FUNCTION_BLOCK FB_T1_InputSource IMPLEMENTS I_InputSource
VAR
	_eDataState: E_DataSourceState;
	
	_nMaxOversamplingFactor: UDINT := 1;
	
	_nElements: UDINT;
	_nCurrentElement: UDINT;
	_nDataHandle: ULINT;
	
	_nClientListHash: LWORD;
	_nCurrentClientHash: LWORD;
	
	_stInputs: ST_T1_Inputs;
	
	fbIotSymbol_GVL_Components_fbMachine_stAnalytics_nState: FB_ALY_IotSymbol_UINT := (stConfig:= (sSymbolName:= 'GVL_Components.fbMachine.stAnalytics.nState'));
	fbIotSymbol_GVL_Components_fbMachine_stAnalytics_nUnitsProduced: FB_ALY_IotSymbol_ULINT := (stConfig:= (sSymbolName:= 'GVL_Components.fbMachine.stAnalytics.nUnitsProduced'));
	fbIotSymbol_GVL_Components_fbMachine_stAnalytics_nDefectiveUnits: FB_ALY_IotSymbol_ULINT := (stConfig:= (sSymbolName:= 'GVL_Components.fbMachine.stAnalytics.nDefectiveUnits'));
	fbIotSymbol_GVL_Components_fbMachine_stAnalytics_tMlCalculation: FB_ALY_IotSymbol_UDINT := (stConfig:= (sSymbolName:= 'GVL_Components.fbMachine.stAnalytics.tMlCalculation'));
	
	//Target T1 = Broker:"localhost" Topic:"DefaultMainTopic/PlcStream1"
	fbStreamHelper: FB_ALY_StreamHelper;
	bConfigured: BOOL := FALSE;
	
	fbTON_DataTimeout: TON;
END_VAR
VAR_STAT
	_nClientIndex: INT;
END_VAR

METHOD AddClient : BOOL
VAR_OUTPUT
	nClientID: LWORD;
END_VAR
VAR
END_VAR
nClientID:= TO_LWORD(EXPT(2,_nClientIndex));
_nClientIndex:= _nClientIndex + 1;

_nClientListHash:= _nClientListHash + nClientID;
END_METHOD

PROPERTY bReadNewData : BOOL
GET
bReadNewData:= _nElements = 0 OR _nCurrentClientHash >= _nClientListHash;
END_GET
END_PROPERTY

METHOD Call : BOOL
VAR
	stConfig: ST_ALY_StreamHelper_Config;
END_VAR
IF NOT fbStreamHelper.bConfigured THEN
	stConfig.nObjectID:= 16#01010110;
	stConfig.nNumInputBuffer:= 20;
	fbStreamHelper.Configure(stConfig);
END_IF

IF NOT bConfigured THEN
	//GVL_Components.fbMachine.stAnalytics.nState
	fbStreamHelper.AddIotSymbol(fbIotSymbol_GVL_Components_fbMachine_stAnalytics_nState);
	//GVL_Components.fbMachine.stAnalytics.nUnitsProduced
	fbStreamHelper.AddIotSymbol(fbIotSymbol_GVL_Components_fbMachine_stAnalytics_nUnitsProduced);
	//GVL_Components.fbMachine.stAnalytics.nDefectiveUnits
	fbStreamHelper.AddIotSymbol(fbIotSymbol_GVL_Components_fbMachine_stAnalytics_nDefectiveUnits);
	//GVL_Components.fbMachine.stAnalytics.tMlCalculation
	fbStreamHelper.AddIotSymbol(fbIotSymbol_GVL_Components_fbMachine_stAnalytics_tMlCalculation);

	bConfigured:= TRUE;
END_IF

fbStreamHelper.Call();
IF fbStreamHelper.bError THEN
	_eDataState:= E_DataSourceState.eError;
ELSIF NOT fbStreamHelper.bConnected THEN
	_eDataState:= E_DataSourceState.eNotConnected;
ELSE
	_nElements:= fbStreamHelper.nNumElements;
	IF _nElements > 0 THEN
		_eDataState:= E_DataSourceState.eReceiveData;
	END_IF

	fbTON_DataTimeout(IN:= _nElements = 0, PT:= T#5S);
	IF fbTON_DataTimeout.Q THEN
		_eDataState:= E_DataSourceState.eWaitForData;
	END_IF
END_IF

IF _nElements > 0 THEN
	_nDataHandle:= _nDataHandle + 1;
	_nCurrentClientHash:= 0;
END_IF

_nCurrentElement:= 0;
END_METHOD

METHOD ClientDone : BOOL
VAR_INPUT
	nClientID: LWORD;
END_VAR
VAR
END_VAR
_nCurrentClientHash:=  _nCurrentClientHash + nClientID;
END_METHOD

PROPERTY eDataState : E_DataSourceState
GET
eDataState:= _eDataState;
END_GET
END_PROPERTY

METHOD GetData : BOOL
VAR_INPUT
	nElement: UDINT;
	pInputs: PVOID;
	nInputsSize: UDINT;
END_VAR
VAR_OUTPUT
	nTimestamp: ULINT;
	nContext: DWORD;
END_VAR
VAR
	_nElement: UDINT;
	_pInputs: PVOID;
	_nInputsSize: UDINT;
END_VAR
Analytics.fbT1_IecCriticalSection.Enter();

_nElement:= nElement;
_pInputs:= pInputs;
_nInputsSize:= nInputsSize;

nContext:= 0;
IF nElements > 0 THEN
	IF _nElement <= nElements THEN

		IF _nCurrentElement <> _nElement THEN

			//Set local raw inputs
			_stInputs.nGVL_Components_fbMachine_stAnalytics_nState:= fbIotSymbol_GVL_Components_fbMachine_stAnalytics_nState.GetValue(_nElement);
			_stInputs.nGVL_Components_fbMachine_stAnalytics_nUnitsProduced:= fbIotSymbol_GVL_Components_fbMachine_stAnalytics_nUnitsProduced.GetValue(_nElement);
			_stInputs.nGVL_Components_fbMachine_stAnalytics_nDefectiveUnits:= fbIotSymbol_GVL_Components_fbMachine_stAnalytics_nDefectiveUnits.GetValue(_nElement);
			_stInputs.nGVL_Components_fbMachine_stAnalytics_tMlCalculation:= fbIotSymbol_GVL_Components_fbMachine_stAnalytics_tMlCalculation.GetValue(_nElement);

			nContext:= E_DataSourceContext.eContext_1000;
			_nCurrentElement:= _nElement;
		END_IF

		//Set output values
		IF _pInputs > 0 THEN
			MEMCPY(_pInputs, ADR(_stInputs), _nInputsSize);
			nTimestamp:= fbStreamHelper.GetTimestampElement(_nElement);
		END_IF
	END_IF
	GetData:= TRUE;
ELSE
	GetData:= FALSE;
END_IF

Analytics.fbT1_IecCriticalSection.Leave();
END_METHOD

PROPERTY nDataHandle : ULINT
GET
nDataHandle:= _nDataHandle;
END_GET
END_PROPERTY

PROPERTY nElements : UDINT
GET
nElements:= _nElements;
END_GET
END_PROPERTY

METHOD NewDataAvailable : BOOL
VAR_INPUT
	nLastDataHandle: ULINT;
END_VAR
VAR
END_VAR
NewDataAvailable:= _nElements > 0 AND _nDataHandle <> nLastDataHandle;
END_METHOD

PROPERTY nMaxOversamplingFactor : UDINT
GET
nMaxOversamplingFactor:= _nMaxOversamplingFactor;
END_GET
END_PROPERTY

END_FUNCTION_BLOCK

(* stored: Version 1.2.0.0, ProductVersion 3.1.4024.13
   POU FB_T1_InputSource: Id {fbbc7d4c-fe99-47a0-a2a3-fc0ec32139bb}, SpecialFunc None
   Folder I_InputSource: Id {e1dcc566-0b00-41ec-a611-4ddb13b5085b}
   Method AddClient: Id {315e74f9-9257-452b-b362-4dc49cf3649a}
   Property bReadNewData: Id {16f7a504-e503-4983-ae04-e5a095d79fa6}
   Get Get: Id {313b3484-4840-44ee-9167-737a8f6a9724}
   Method Call: Id {ca01f449-2322-4938-8163-f106edd3b239}
   Method ClientDone: Id {bf19a8bd-b79f-4a04-9aa1-24abf9ac7972}
   Property eDataState: Id {ed605f32-b43d-4e05-86d6-4d04f9981256}
   Get Get: Id {12dd5f27-34f0-4511-952e-87b7af302fc7}
   Method GetData: Id {d6e405cd-3e34-4ed6-96af-d68922a35077}
   Property nDataHandle: Id {25b8829c-9b48-4dc3-8882-fe2283e3cf6c}
   Get Get: Id {685394dd-f868-4dd6-8daa-0f7bdd5b38e9}
   Property nElements: Id {3e736a4f-1557-46ba-b541-eaec3d098b7a}
   Get Get: Id {2b573a8b-5de9-418d-9d2c-5010798406d1}
   Method NewDataAvailable: Id {4847d983-5d67-4dc7-921e-5497973d374e}
   Property nMaxOversamplingFactor: Id {788fabef-a447-4ace-84d4-c022167150a2}
   Get Get: Id {d81778d6-ad07-417d-b841-cec93d912d67} *)
